{attribute 'TcGenerated'}
{attribute 'no-analysis'}
{attribute 'linkalways'}
// This function has been automatically generated from the project information.
VAR_GLOBAL CONSTANT
	{attribute 'const_non_replaced'}
	stLibVersion_Xts_Library : ST_LibVersion := (iMajor := 16, iMinor := 0, iBuild := 2, iRevision := 0, nFlags := 1, sVersion := '16.0.2');
END_VAR

(* stored: Version 1.1.0.1
   GVL Global_Version: Id {e78b1c7b-fbdf-486e-ac70-aee233bacb57} *)
